KUKA KRL data list: TestBaseCalc.dat

&ACCESS RVO1
DEFDAT  TESTBASECALC PUBLIC

GLOBAL FRAME testBase={X -0.758253098,Y -1.00336087,Z 5.00191593,A -0.0486980379,B 0.0257083867,C -0.0256476030}
ENDDAT
